FUNCTION_BLOCK FB_S1_Sequence
VAR_INPUT
	SFCinit:BOOL;
END_VAR
VAR_OUTPUT
END_VAR
VAR
END_VAR

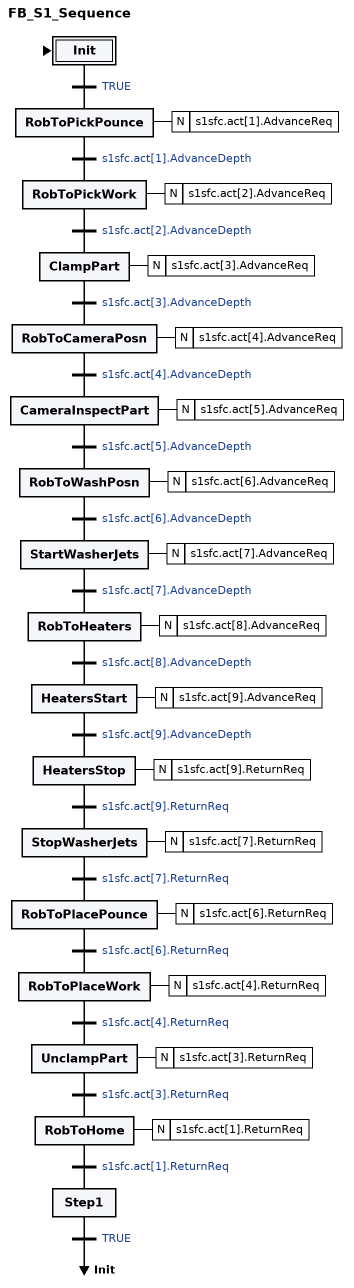
INITIAL_STEP Init:
END_STEP
TRANSITION FROM Init TO RobToPickPounce
    := TRUE;
END_TRANSITION
STEP RobToPickPounce:
    s1sfc.act[1].AdvanceReq(N);
END_STEP
TRANSITION FROM RobToPickPounce TO RobToPickWork
    := s1sfc.act[1].AdvanceDepth;
END_TRANSITION
STEP RobToPickWork:
    s1sfc.act[2].AdvanceReq(N);
END_STEP
TRANSITION FROM RobToPickWork TO ClampPart
    := s1sfc.act[2].AdvanceDepth;
END_TRANSITION
STEP ClampPart:
    s1sfc.act[3].AdvanceReq(N);
END_STEP
TRANSITION FROM ClampPart TO RobToCameraPosn
    := s1sfc.act[3].AdvanceDepth;
END_TRANSITION
STEP RobToCameraPosn:
    s1sfc.act[4].AdvanceReq(N);
END_STEP
TRANSITION FROM RobToCameraPosn TO CameraInspectPart
    := s1sfc.act[4].AdvanceDepth;
END_TRANSITION
STEP CameraInspectPart:
    s1sfc.act[5].AdvanceReq(N);
END_STEP
TRANSITION FROM CameraInspectPart TO RobToWashPosn
    := s1sfc.act[5].AdvanceDepth;
END_TRANSITION
STEP RobToWashPosn:
    s1sfc.act[6].AdvanceReq(N);
END_STEP
TRANSITION FROM RobToWashPosn TO StartWasherJets
    := s1sfc.act[6].AdvanceDepth;
END_TRANSITION
STEP StartWasherJets:
    s1sfc.act[7].AdvanceReq(N);
END_STEP
TRANSITION FROM StartWasherJets TO RobToHeaters
    := s1sfc.act[7].AdvanceDepth;
END_TRANSITION
STEP RobToHeaters:
    s1sfc.act[8].AdvanceReq(N);
END_STEP
TRANSITION FROM RobToHeaters TO HeatersStart
    := s1sfc.act[8].AdvanceDepth;
END_TRANSITION
STEP HeatersStart:
    s1sfc.act[9].AdvanceReq(N);
END_STEP
TRANSITION FROM HeatersStart TO HeatersStop
    := s1sfc.act[9].AdvanceDepth;
END_TRANSITION
STEP HeatersStop:
    s1sfc.act[9].ReturnReq(N);
END_STEP
TRANSITION FROM HeatersStop TO StopWasherJets
    := s1sfc.act[9].ReturnReq;
END_TRANSITION
STEP StopWasherJets:
    s1sfc.act[7].ReturnReq(N);
END_STEP
TRANSITION FROM StopWasherJets TO RobToPlacePounce
    := s1sfc.act[7].ReturnReq;
END_TRANSITION
STEP RobToPlacePounce:
    s1sfc.act[6].ReturnReq(N);
END_STEP
TRANSITION FROM RobToPlacePounce TO RobToPlaceWork
    := s1sfc.act[6].ReturnReq;
END_TRANSITION
STEP RobToPlaceWork:
    s1sfc.act[4].ReturnReq(N);
END_STEP
TRANSITION FROM RobToPlaceWork TO UnclampPart
    := s1sfc.act[4].ReturnReq;
END_TRANSITION
STEP UnclampPart:
    s1sfc.act[3].ReturnReq(N);
END_STEP
TRANSITION FROM UnclampPart TO RobToHome
    := s1sfc.act[3].ReturnReq;
END_TRANSITION
STEP RobToHome:
    s1sfc.act[1].ReturnReq(N);
END_STEP
TRANSITION FROM RobToHome TO Step1
    := s1sfc.act[1].ReturnReq;
END_TRANSITION
STEP Step1:
END_STEP
TRANSITION FROM Step1 TO Init
    := TRUE;
END_TRANSITION

END_FUNCTION_BLOCK

(* stored: Version 1.1.0.1, ProductVersion 3.1.4024.12
   POU FB_S1_Sequence: Id {0e1c489b-0d88-4453-80c3-4355fd852980}, SpecialFunc None *)
